(* Logix 5000 project; controller Hoa_Example Emulate 5570 rev 20.11; software revision 20.00 *)

TASK MainTask (continuous, watchdog 500 ms) : MainProgram

MODULES
   Local : Emulate 5570 (ICP 1, rev 20.11)
END_MODULES

PROGRAM MainProgram   (* main routine _00_Main *)
VAR
   Blower_En : BOOL; {access Read Only}
   Blower_PB_Auto : BOOL; {access Read Only}
   Blower_PB_Hand : BOOL; {access Read Only}
   Blower_PB_Off : BOOL; {access Read Only}
   Hoa_Mode : DINT; {access Read Only}   // 0: Hand Mode 1: Off Mode 2: Auto Mode
   IN_PB_AUTO : BOOL; {access Read Only}
   IN_PB_HAND : BOOL; {access Read Only}
   IN_PB_OFF : BOOL; {access Read Only}
   OUT_PB_BLOWER_EN : BOOL; {access Read Only}
END_VAR

ROUTINE _00_Main   (* ladder *)
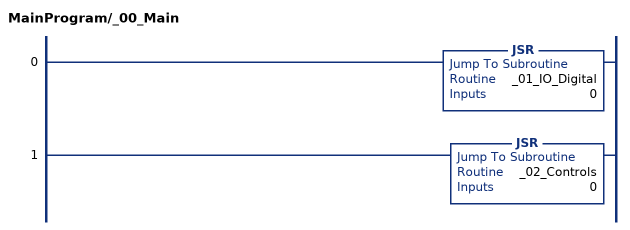
   0: JSR(_01_IO_Digital,0);
   1: JSR(_02_Controls,0);
END_ROUTINE

ROUTINE _01_IO_Digital   (* ladder *)
// Digital IO
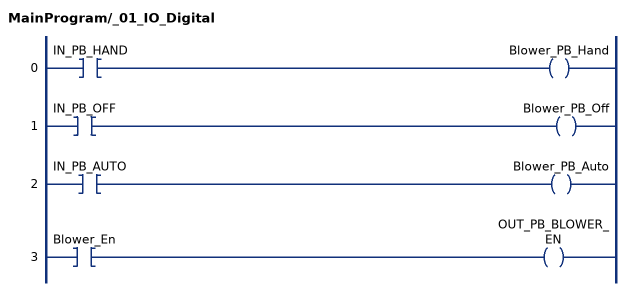
   0: XIC(IN_PB_HAND)OTE(Blower_PB_Hand);
   1: XIC(IN_PB_OFF)OTE(Blower_PB_Off);
   2: XIC(IN_PB_AUTO)OTE(Blower_PB_Auto);
   3: XIC(Blower_En)OTE(OUT_PB_BLOWER_EN);
END_ROUTINE

ROUTINE _02_Controls   (* ladder *)
// Controls
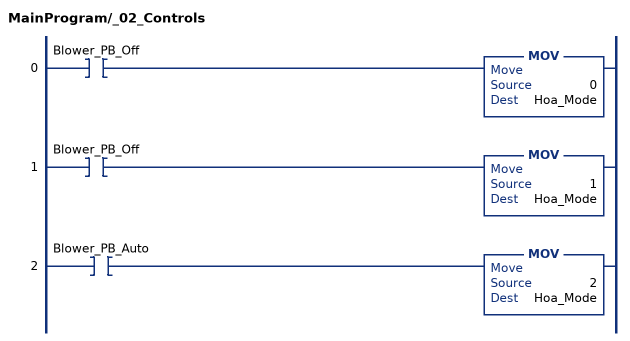
   0: XIC(Blower_PB_Off)MOV(0,Hoa_Mode);
   1: XIC(Blower_PB_Off)MOV(1,Hoa_Mode);
   2: XIC(Blower_PB_Auto)MOV(2,Hoa_Mode);
END_ROUTINE
END_PROGRAM
